(* IEC 61131-3 sources: SmartHomeNew/snapshots/project_clean_state_2026_04_16/workspace/dut_rebuild/dhw_v2/extraction, 2 files *)

(* ---- FB_DHW_Command_Extractor_DRAFT.st ---- *)
FUNCTION_BLOCK FB_DHW_Command_Extractor_DRAFT
VAR_INPUT
    VI_Enable : BOOL;
    VI_Target_Temp : REAL;
END_VAR
VAR_OUTPUT
    VO_Command : ST_DHW_Command_V2;
END_VAR

VO_Command.Enabled := VI_Enable;
VO_Command.Target_Temp := VI_Target_Temp;
END_FUNCTION_BLOCK

(* ---- FB_DHW_State_Extractor_DRAFT.st ---- *)
FUNCTION_BLOCK FB_DHW_State_Extractor_DRAFT
VAR_INPUT
    VI_Tank_Temp : REAL;
END_VAR
VAR_OUTPUT
    VO_State : ST_DHW_State_V2;
END_VAR

VO_State.Tank_Temp := VI_Tank_Temp;
END_FUNCTION_BLOCK
